{attribute 'qualified_only'}
//{attribute 'strict'}
{attribute 'to_string'}
TYPE nChiniseMachineErrorCodes :
(
	// Błędy ogólne
	NoError := 0,
	UnKnownAlarm := 53,						// Niezidentyfikowany alarm maszyny
	UnKnownLock := 54,						// Niezidentyfikowana blokada maszyny
	ResetTimeout := 518,					// Timeout resetu maszyny
	ProgramConfigError := 90,				// Błąd w konfiguracji programu
	SafetySystemNotArmed := 614,			// System safety nie uzbrojony
	NoMachineReactionOnStartSig := 140,		// Brak reakcji na sygnał startu (brak wysunięcia siłownika - brak powietrza itp.)


	
	MemoryError 		:= 1,
	RTC_error 			:= 2,
	HomePositionError 	:= 3,
	TriggerPointError 	:= 4,
	PressureError 		:= 5,
	FrequencyError 		:= 6,
	TimeErrorMin 		:= 7,
	TimeErrorMax 		:= 8,
	EnergyErrorMin 		:= 9,
	EnergyErrorMax 		:= 10,
	PowerErrorMin 		:= 11,
	PowerErrorMax 		:= 12,
	DRM_errorMin 		:= 13,
	DRM_errorMax 		:= 14,
	ABS_errorMin  		:= 15,
	ABS_errorMax  		:= 16,
	MonitTimeExpired 	:= 17,
	NoUltrasound 		:= 18,
	WP_AUX1_Error 		:= 19,
	WP_AUX2_Error 		:= 20,
	HP_AUX1_Error 		:= 21,
	HP_AUX2_Error 		:= 22,
	EmergencyStop 		:= 23,
	ResetIsPressed 		:= 24,
	MemCodingError 		:= 25,
	CondAUX1_Error 		:= 26,
	CondAUX2_Error 		:= 27,
	RewinderError 		:= 28,
	GenCommError 		:= 29,
	ExceedTemperature 	:= 30,
	ExceedProtection 	:= 31,
	GeneratorError 		:= 32,
	ActiveCurtain 		:= 33,
	StartSgnError 		:= 34,
	PowerSupplyError 	:= 35,
	EncoderError 		:= 36,
	ProgramError 		:= 37,
	ParametersError 	:= 38,
	MeasurementError 	:= 39,
	ProgSelError 		:= 40,
	WrongSocket 		:= 41,
	GenModeError 		:= 42,
	GenEnergyError 		:= 43,
	GenPowerError 		:= 44,
	GenParamError 		:= 45,
	NoTransducer 		:= 46,
	GenMultiResonance 	:= 47,
	GenDuringScan  		:= 48,
	ProgGenError 		:= 49,
	SkanGenError 		:= 50,
	Communication_error := 51,
	UndefinedError		:= 52,
	FixtureNoResponse	:= 55,
	FixtureError		:= 57,
	BreakStartSignal 	:= 127,
	SendFrameError		:= 128,
	AUX1OutNotSetUp		:= 129,
	StartSignalToShort 	:= 191,
		
	OutputErrorWeldOk 	:= 86,
	OutputErrorReady 	:= 87,
	OutputErrorError 	:= 88,
	ExtCondNotMet		:= 92,
	communicationError := 999
);
END_TYPE

(* stored: Version 1.1.0.1, ProductVersion 3.1.4024.13
   EnumerationTextList nChiniseMachineErrorCodes: Id {da1fdd11-04d2-4a70-8407-844f1a8461ec} *)
